PROGRAM pouDataDisplay
VAR
	FB_DataCombine_0: FB_DataCombine;
	FB_DataCombine_1: FB_DataCombine;
	FB_DataCombine_2: FB_DataCombine;
	FB_DataCombine_3: FB_DataCombine;
	FB_DataCombine_4: FB_DataCombine;
	FB_DataCombine_5: FB_DataCombine;
	FB_DataCombine_6: FB_DataCombine;
	FB_DataCombine_7: FB_DataCombine;
	FB_DataCombine_8: FB_DataCombine;
	FB_DataCombine_9: FB_DataCombine;
	FB_DataCombine_10: FB_DataCombine;
	FB_DataCombine_11: FB_DataCombine;
	FB_DataCombine_12: FB_DataCombine;
	FB_DataCombine_13: FB_DataCombine;
	FB_DataCombine_14: FB_DataCombine;
	FB_DataCombine_16: FB_DataCombine;
	werd: DWORD;
END_VAR

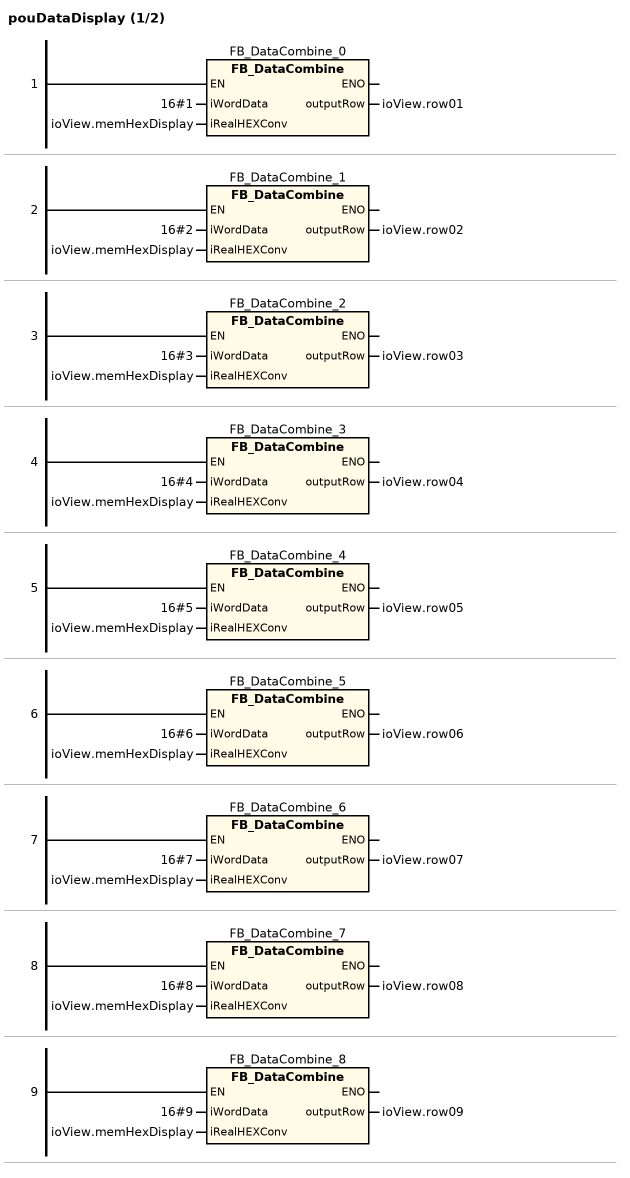
// NETWORK 1
FB_DataCombine_0(iWordData := 16#1, iRealHEXConv := ioView.memHexDisplay, outputRow => ioView.row01); // FB_DataCombine

// NETWORK 2
FB_DataCombine_1(iWordData := 16#2, iRealHEXConv := ioView.memHexDisplay, outputRow => ioView.row02); // FB_DataCombine

// NETWORK 3
FB_DataCombine_2(iWordData := 16#3, iRealHEXConv := ioView.memHexDisplay, outputRow => ioView.row03); // FB_DataCombine

// NETWORK 4
FB_DataCombine_3(iWordData := 16#4, iRealHEXConv := ioView.memHexDisplay, outputRow => ioView.row04); // FB_DataCombine

// NETWORK 5
FB_DataCombine_4(iWordData := 16#5, iRealHEXConv := ioView.memHexDisplay, outputRow => ioView.row05); // FB_DataCombine

// NETWORK 6
FB_DataCombine_5(iWordData := 16#6, iRealHEXConv := ioView.memHexDisplay, outputRow => ioView.row06); // FB_DataCombine

// NETWORK 7
FB_DataCombine_6(iWordData := 16#7, iRealHEXConv := ioView.memHexDisplay, outputRow => ioView.row07); // FB_DataCombine

// NETWORK 8
FB_DataCombine_7(iWordData := 16#8, iRealHEXConv := ioView.memHexDisplay, outputRow => ioView.row08); // FB_DataCombine

// NETWORK 9
FB_DataCombine_8(iWordData := 16#9, iRealHEXConv := ioView.memHexDisplay, outputRow => ioView.row09); // FB_DataCombine

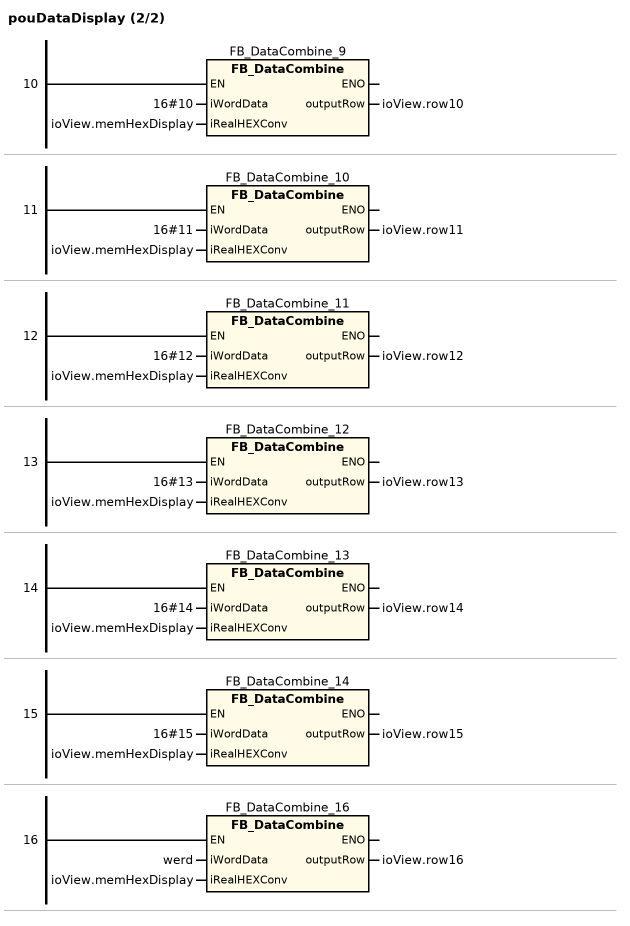
// NETWORK 10
FB_DataCombine_9(iWordData := 16#10, iRealHEXConv := ioView.memHexDisplay, outputRow => ioView.row10); // FB_DataCombine

// NETWORK 11
FB_DataCombine_10(iWordData := 16#11, iRealHEXConv := ioView.memHexDisplay, outputRow => ioView.row11); // FB_DataCombine

// NETWORK 12
FB_DataCombine_11(iWordData := 16#12, iRealHEXConv := ioView.memHexDisplay, outputRow => ioView.row12); // FB_DataCombine

// NETWORK 13
FB_DataCombine_12(iWordData := 16#13, iRealHEXConv := ioView.memHexDisplay, outputRow => ioView.row13); // FB_DataCombine

// NETWORK 14
FB_DataCombine_13(iWordData := 16#14, iRealHEXConv := ioView.memHexDisplay, outputRow => ioView.row14); // FB_DataCombine

// NETWORK 15
FB_DataCombine_14(iWordData := 16#15, iRealHEXConv := ioView.memHexDisplay, outputRow => ioView.row15); // FB_DataCombine

// NETWORK 16
FB_DataCombine_16(iWordData := werd, iRealHEXConv := ioView.memHexDisplay, outputRow => ioView.row16); // FB_DataCombine

END_PROGRAM

(* stored: Version 1.1.0.1, ProductVersion 3.1.4024.12
   POU pouDataDisplay: Id {9d244046-dbb0-4950-8033-df6cea4a2323}, SpecialFunc None *)
